PROGRAM MAIN
VAR
	nCounter : INT := 0;
	nCounter3 : INT := 0;
END_VAR

nCounter:= nCounter + 1;
nCounter3:= nCounter + 10;

END_PROGRAM

(* stored: Version 1.1.0.1, ProductVersion 3.1.4024.12
   POU MAIN: Id {6f1433b0-af06-4830-84af-256fba9d2b49}, SpecialFunc None *)
